// TwinCAT 3 PLC project utils
// Title: ESO ELT Utility Library
// Company: ESO
// Author: Mario Kiekebusch
// ProjectVersion: 0.0.0.2
// Description: ELT - Library provide general purpose utilities.
// ProgramVersion: 3.1.4023.0
// libraries:
//   ESO LDC Common Library, * (ESO)
//   ESO LDC Timer Library, * (ESO)
//   ESO MUDPI Library, * (ESO)
//   Tc2_Standard, * (Beckhoff Automation GmbH)
//   Tc2_System, * (Beckhoff Automation GmbH)
//   Tc2_Utilities, * (Beckhoff Automation GmbH)
//   Tc3_EventLogger, * (Beckhoff Automation GmbH)
//   Tc3_Module, * (Beckhoff Automation GmbH)
//   VisuDialogs, * (System)
// project tree:
//   DUTs/Structures/ T_EVENTLOG_PAYLOAD.TcDUT, T_EVENT_PUB_ELEM.TcDUT, T_IP_ADDRESS.TcDUT, T_PACKET_INFO.TcDUT, T_UDP_INFO.TcDUT
//   / GlobalTextList.TcGTLO, PlcTask.TcTTO, Visualization Manager.TcVMO (not stored)
//   GVLs/ GVL.TcGVL
//   POUs/ FB_DataSetFifo.TcPOU, FB_EVENT_LISTENER.TcPOU, FB_MUDPI_RECEIVER.TcPOU, FB_MUDPI_SENDER.TcPOU, FB_SAMPLE_LISTENER.TcPOU, MAIN.TcPOU
//   Version/ Global_Version.TcGVL
//   VISUs/Templates/ GUI_TEMPLATE_MUDPI_RECEIVER.TcVIS, GUI_TEMPLATE_MUDPI_SENDER.TcVIS
// real-time tasks:
//   TASK PlcTask: cycle T#10ms, priority 20, ADS port 350

CONFIGURATION utils
    RESOURCE PLC ON TwinCAT3
        TASK PlcTask(INTERVAL := T#10ms, PRIORITY := 20);
        PROGRAM MAIN WITH PlcTask : MAIN;
    END_RESOURCE
END_CONFIGURATION

// ---- DUTs/Structures/T_EVENTLOG_PAYLOAD.TcDUT
TYPE T_EVENTLOG_PAYLOAD :
STRUCT
	{attribute 'TcEncoding':='UTF-8'}
	source : STRING(80) := ''; 
	severity : INT := 0; 
	{attribute 'TcEncoding':='UTF-8'}
	text: STRING(255) := '';
	timestamp: ULINT;
END_STRUCT
END_TYPE

// ---- DUTs/Structures/T_EVENT_PUB_ELEM.TcDUT
TYPE T_EVENT_PUB_ELEM :
STRUCT
	fbEventText: FB_RequestEventText;
	bTextRequest: BOOL := FALSE;
	payload: T_EVENTLOG_PAYLOAD;
END_STRUCT
END_TYPE

// ---- DUTs/Structures/T_IP_ADDRESS.TcDUT
TYPE T_IP_ADDRESS :
UNION
	ipAdrInternal : UDINT;
	ipAdr : ARRAY[0..3] OF BYTE;
END_UNION
END_TYPE

// ---- DUTs/Structures/T_PACKET_INFO.TcDUT
TYPE T_PACKET_INFO :
STRUCT
	topicId: UDINT; 
	componentId: UINT; // counter the number of times the diagnostic data was sent.
	sampleId: UDINT; 
	frameId: UINT;
	numFrames: UINT;
	version: UINT;
	appTag: UINT;
	timestamp: LREAL;
	payloadSize: UINT;	
	size: UINT;
	valid: BOOL;
END_STRUCT
END_TYPE

// ---- DUTs/Structures/T_UDP_INFO.TcDUT
TYPE T_UDP_INFO :
STRUCT
	bDriverInitialization: BOOL; // Indication of whether the realtime driver is properly initialized.  
	nReceivedPackets: UDINT; // counter the number of times the diagnostic data was sent.
	uSenderAddress: T_IP_ADDRESS;
	ipv4Adr : T_IPv4Addr := '';
	lrNotification: LREAL; // timestamp of the last sent
	sNotification: STRING;
END_STRUCT
END_TYPE

// ---- GVLs/GVL.TcGVL
VAR_GLOBAL CONSTANT
	MAX_BUFFER_SIZE : UDINT := 35000;
	MAX_EVENTS_SIZE : INT := 100;
END_VAR

// ---- Version/Global_Version.TcGVL
{attribute 'TcGenerated'}
{attribute 'no-analysis'}
{attribute 'linkalways'}
// This function has been automatically generated from the project information.
VAR_GLOBAL CONSTANT
	{attribute 'const_non_replaced'}
	stLibVersion_ESO_ELT_Utility_Library : ST_LibVersion := (iMajor := 0, iMinor := 0, iBuild := 0, iRevision := 2, nFlags := 0, sVersion := '0.0.0.2');
END_VAR

// ---- POUs/MAIN.TcPOU
PROGRAM MAIN
VAR
END_VAR

END_PROGRAM

// ---- POUs/FB_DataSetFifo.TcPOU
FUNCTION_BLOCK FB_DataSetFifo
VAR_INPUT
	bOverwrite	: BOOL;
	in 			: T_EVENTLOG_PAYLOAD;
END_VAR
VAR_OUTPUT
	bOk			: BOOL;
	nCount		: UDINT;
	nLoad		: UDINT;
	out			: T_EVENTLOG_PAYLOAD;
END_VAR
VAR
	arrBuffer 	: ARRAY[0..MAX_BUFFER_SIZE] OF BYTE; (* Buffer memory used by FB_MemRingBuffer function block *)
	fbBuffer	: FB_MemRingBuffer;
	dataset_size: UDINT;
END_VAR

;

ACTION A_Add:
fbBuffer.A_AddTail( pWrite:= ADR( in ),
					cbWrite:= SIZEOF( in ),
					pBuffer:= ADR( arrBuffer ),
					cbBuffer:= SIZEOF( arrBuffer ),
					bOk=> bOk,
					nCount => nCount );


IF NOT bOk THEN (* overflow ? *)
	IF bOverwrite THEN
		fbBuffer.A_RemoveHead(); (* remove one oldest entry *)

		fbBuffer.A_AddTail( bOk => bOk, nCount => nCount );
	END_IF
END_IF


dataset_size := SIZEOF(in);
nLoad := (fbBuffer.cbSize * 100) / MAX_BUFFER_SIZE;
END_ACTION

ACTION A_Get:
fbBuffer.A_GetHead( pRead:= ADR( out ),
					cbRead:= SIZEOF( out ),
					pBuffer:= ADR( arrBuffer ),
					cbBuffer:= SIZEOF( arrBuffer ),
					bOk=> bOk,
					nCount => nCount );

nLoad := (fbBuffer.cbSize * 100) / MAX_BUFFER_SIZE;
END_ACTION

ACTION A_Remove:
fbBuffer.A_RemoveHead( 	pRead:= ADR( out ),
						cbRead:= SIZEOF( out ),
						pBuffer:= ADR( arrBuffer ),
						cbBuffer:= SIZEOF( arrBuffer ),
						bOk=> bOk,
						nCount => nCount );

nLoad := (fbBuffer.cbSize * 100) / MAX_BUFFER_SIZE;
END_ACTION

ACTION A_Reset:
MEMSET( ADR( arrBuffer ), 0, SIZEOF( arrBuffer ) ); (* reset (optional) internal buffer *)

fbBuffer.A_Reset( 	bOk=> bOk,
					nCount => nCount );

nLoad := (fbBuffer.cbSize * 100) / MAX_BUFFER_SIZE;
END_ACTION

METHOD IsEmpty : BOOL
VAR_INPUT
END_VAR
IF nCount > 0 THEN
	IsEmpty := FALSE;
	RETURN;
END_IF

IsEmpty := TRUE;
return;
END_METHOD

METHOD Size : UDINT
VAR_INPUT
END_VAR
Size := nCount;
END_METHOD

END_FUNCTION_BLOCK

// ---- POUs/FB_EVENT_LISTENER.TcPOU
FUNCTION_BLOCK FB_EVENT_LISTENER
VAR_INPUT
	refFbEventFilter  : REFERENCE TO FB_TcEventFilter; 
	refFbTime:  REFERENCE TO FB_TIME;
END_VAR
VAR_OUTPUT
END_VAR
VAR
	hr : HRESULT;
	
	bSubscribe : BOOL := TRUE;
	bSubscribed : BOOL;
	bUnSubscribe : BOOL;
	
	fbMessageListener : FB_SAMPLE_LISTENER;
	Message: INT;
	
END_VAR

fbMessageListener.CustomExecute(refFbTime); // retrieve messages and its texts


IF bSubscribe THEN 
	bSubscribe := FALSE;
	hr := fbMessageListener.Subscribe2(refFbEventFilter); //subscribe to retrieve defined events
	IF SUCCEEDED(hr) THEN	
		bSubscribed := TRUE;
	END_IF
END_IF 

IF bUnSubscribe THEN 
	bUnSubscribe := FALSE;
	hr := fbMessageListener.Unsubscribe();
	IF SUCCEEDED(hr) THEN	
		bSubscribed := FALSE;
	END_IF
END_IF

END_FUNCTION_BLOCK

// ---- POUs/FB_SAMPLE_LISTENER.TcPOU
FUNCTION_BLOCK FB_SAMPLE_LISTENER EXTENDS FB_ListenerBase2
VAR_INPUT
END_VAR
VAR_OUTPUT
END_VAR
VAR
	sJsonAttribute : STRING (10000);	
	hr : HRESULT;
	
	nCntMessagesSent : INT;
	nCntAlarmsRaised : INT;
	nCntAlarmsConfirmed : INT;
	nCntAlarmsCleared : INT;
	
	fbSender: FB_MUDPI_SENDER;
	arrEvents : ARRAY[0..MAX_EVENTS_SIZE] OF T_EVENT_PUB_ELEM;
	nCntEventReceived : INT := 0;
	fbFifo 		: FB_DataSetFifo := ( bOverwrite := TRUE );
	newEntry	: T_EVENTLOG_PAYLOAD;
	oldEntry	: T_EVENTLOG_PAYLOAD;
	bSuccess	: BOOL;
	nCount		: UDINT;
	nLoad		: UDINT;
	nWaitCounter : UDINT := 0;
END_VAR

METHOD CustomExecute : HRESULT
VAR_INPUT
	refFbTime:  REFERENCE TO FB_TIME;
END_VAR

VAR
	hr : HRESULT;
	counter: INT := 0;
END_VAR
hr := SUPER^.Execute(); //retrieve events
fbSender();
(* Go through the list of buffers to check if there new events *)
FOR counter := 0 TO MAX_EVENTS_SIZE BY 1 DO
	IF arrEvents[counter].bTextRequest THEN
		IF arrEvents[counter].fbEventText.bError THEN
			arrEvents[counter].payload.text := 'Error';
			arrEvents[counter].bTextRequest := FALSE;
			fbFifo.A_Add(	in := arrEvents[counter].payload, bOk=>bSuccess, nCount=> nCount, nLoad => nLoad );
		ELSIF NOT arrEvents[counter].fbEventText.bBusy THEN
			arrEvents[counter].fbEventText.GetString(arrEvents[counter].payload.text, SIZEOF(arrEvents[counter].payload.text));
			arrEvents[counter].bTextRequest := FALSE;
			(* add new entry to the fifo *)
			fbFifo.A_Add(	in := arrEvents[counter].payload, bOk=>bSuccess, nCount=> nCount, nLoad => nLoad );
		END_IF
	END_IF
END_FOR

// Forces to send one log per every ten cycles.
// Due to the asynchronous nature of the TC Event Logging, sending the logs faster has 
// shown some problems. 
IF NOT fbFifo.IsEmpty() THEN
	nWaitCounter := nWaitCounter + 1;
	IF nWaitCounter > 10 THEN
		(* remove oldest entry from them ring buffer*)
		fbFifo.A_Remove( out => oldEntry, bOk => bSuccess, nCount => nCount, nLoad => nLoad );
		IF bSuccess THEN
			(* Send log info *)
			fbSender.SetTimestamp(refFbTime.GetMudpiTime());
			fbSender.SetMudpiPayload(ADR(oldEntry), SIZEOF(oldEntry));
			fbSender.SendData();
			(* Reset counter *)
			nWaitCounter := 0;
		END_IF
	END_IF
END_IF 



CustomExecute:= hr;
END_METHOD

METHOD OnAlarmCleared : HRESULT
VAR_INPUT
	fbEvent : REFERENCE TO FB_TcEvent;
END_VAR
nCntAlarmsCleared := nCntAlarmsCleared + 1;

OnAlarmCleared := S_OK; // in order to receive more callbacks (Set <> S_OK in order to cancel the callbacks for this program cycle.)
END_METHOD

METHOD OnAlarmConfirmed : HRESULT
VAR_INPUT
	fbEvent : REFERENCE TO FB_TcEvent;
END_VAR
nCntAlarmsConfirmed := nCntAlarmsConfirmed + 1;

OnAlarmConfirmed := S_OK; // in order to receive more callbacks (Set <> S_OK in order to cancel the callbacks for this program cycle.)
END_METHOD

METHOD OnAlarmRaised : HRESULT
VAR_INPUT
	fbEvent : REFERENCE TO FB_TcEvent;
END_VAR
hr := fbEvent.GetJsonAttribute(sJsonAttribute, SIZEOF(sJsonAttribute));
nCntAlarmsRaised := nCntAlarmsRaised + 1;

OnAlarmRaised := S_OK; // in order to receive more callbacks (Set <> S_OK in order to cancel the callbacks for this program cycle.)
END_METHOD

METHOD OnMessageSent : HRESULT
VAR_INPUT
	fbEvent : REFERENCE TO FB_TcEvent;
END_VAR

VAR
	payload: T_EVENTLOG_PAYLOAD;
	fbRequestEventText : FB_RequestEventText;
END_VAR
hr := fbEvent.GetJsonAttribute(sJsonAttribute, SIZEOF(sJsonAttribute));

(* Store events in an array since they could arrive in bursts *)
arrEvents[nCntEventReceived].bTextRequest :=  TRUE;
arrEvents[nCntEventReceived].payload.source := fbEvent.ipSourceInfo.sName;
arrEvents[nCntEventReceived].payload.severity := fbEvent.eSeverity;
arrEvents[nCntEventReceived].payload.timestamp := fbEvent.nTimestamp;
arrEvents[nCntEventReceived].fbEventText.Request(eventClass:=fbEvent.EventClass, nEventId:=fbEvent.nEventId, nLangId:=1033, ipArgs:=fbEvent.ipArguments );
arrEvents[nCntEventReceived].bTextRequest :=  TRUE;
nCntMessagesSent := nCntMessagesSent + 1;
nCntEventReceived := nCntEventReceived + 1;
(*
If number of events are bigger than the buffer size, start overiding 
The risk of loosing events is low since we have a ring buffer storing 
the events to be sent outside. 
*)
IF nCntEventReceived >= MAX_EVENTS_SIZE THEN
	nCntEventReceived := 0;
END_IF



OnMessageSent := S_OK; // in order to receive more callbacks (Set <> S_OK in order to cancel the callbacks for this program cycle.)
END_METHOD

END_FUNCTION_BLOCK

// ---- POUs/FB_MUDPI_SENDER.TcPOU
(*
    This function blocks aims to pack the EL6688 diagnostic data in MUDPI frames
    and transmit them to Time System using Beckhoffs realtime UDP driver (TF6311). 
    The user of this function blocks needs to do the following in order for the library to work correctly:
    - Initialize the library with configuration parameters
        - Destination IP-address (a multicast address)
        - Destination port
        - Source port
*)

{attribute 'c++_compatible'}
FUNCTION_BLOCK FB_MUDPI_SENDER IMPLEMENTS ITcIoUdpProtocolRecv
VAR_INPUT
		ipAddress : Tc2_System.T_IPv4Addr := '0.0.0.0';
		dest_port : UINT := 10000;
		local_port : UINT := 20000;
		instance_name: STRING := 'undefined';
END_VAR
VAR_OUTPUT
END_VAR
VAR
	(* TF6311 realtime driver parameters *)
    {attribute 'TcInitSymbol'}
    oid : OTCID;
    ipUdp : ITcIoUdpProtocol;
    nReceivedPackets : UINT;
    uLastReceivedIP : T_IP_ADDRESS;
    hrInit : HRESULT;
    hrSend : HRESULT; 
    bSuccessfulInitializationOfRealtimeDriver : BOOL := FALSE; // Indication of whether the realtime driver is properly initialized.
	bEnableSending : BOOL := FALSE; // Indication of whether the sender is active or not.
	
	mudpiPacket : ESO_MUDPI.FB_MudpiPacket(topicId := 300, componentId := 5);
	packet_info : T_PACKET_INFO;
	
	  (* Transmission/communication parameters *)
	_destinationIpAddressString : Tc2_System.T_IPv4Addr;
    _destinationIpAddress : UDINT; // Destination address for the data
    _destinationPort : UINT; // Destination port for the data
    _sourcePort : UINT; // Source port of the data
	
	sLibVersion:	   STRING	:= 'UNKNOWN'; // Library version
	
END_VAR

(*
_destinationIpAddressString := ipAddress;
_destinationPort := dest_port;
_sourcePort := local_port;
*)

IF ipUdp <> 0 THEN
	ipUdp.CheckReceived();
END_IF

UpdateMudpiPacket();

METHOD FB_exit : BOOL
VAR_INPUT
    bInCopyCode : BOOL; // if TRUE, the exit method is called for exiting an instance that is copied afterwards (online change).
END_VAR
IF NOT bInCopyCode THEN // no online change
    IF ipUdp <> 0 THEN
        //ipUdp.UnregisterReceiver(nUdpPort); // Shutdown
        //ipUdp.UnregisterReceiver(nUdpPort); // Shutdown
        FW_SafeRelease(ADR(ipUdp));
        FB_exit := TRUE;
    END_IF
END_IF
END_METHOD

METHOD FB_init : BOOL
VAR_INPUT
    bInitRetains : BOOL; // if TRUE, the retain variables are initialized (warm start / cold start)
    bInCopyCode : BOOL;  // if TRUE, the instance afterwards gets moved into the copy code (online change)
END_VAR

sLibVersion := stLibVersion_ESO_ELT_Utility_Library.sVersion;
_destinationIpAddressString := ipAddress;
_destinationPort := dest_port;
_sourcePort := local_port;

IF NOT bInCopyCode THEN // no online change
	IF ipUdp = 0 AND oid <> 0 THEN
	    hrInit := FW_ObjMgr_GetObjectInstance(	oid:=oid, 
											iid:=TC_GLOBAL_IID_LIST.IID_ITcIoUdpProtocol, 
											pipUnk:=ADR(ipUdp) );
		
		IF SUCCEEDED(hrInit) THEN 
			bSuccessfulInitializationOfRealtimeDriver := TRUE;
		(*
			IF  SUCCEEDED(ipUdp.RegisterReceiver(nUdpPort, THIS^)) THEN //open port
				FB_init := TRUE;
			ELSE 
				FB_init := FALSE; 
				FW_SafeRelease(ADR(ipUdp));
			END_IF
			*)
		END_IF
		
	ELSIF oid = 0 THEN 
		FB_init := FALSE; 
		hrInit := ERR_INVALID_PARAM; 				
	END_IF
END_IF
END_METHOD

METHOD FB_reinit : BOOL
IF (ipUdp <> 0) THEN
    //ipUdp.RegisterReceiver(nUdpPort, THIS^);
    //ipUdp.RegisterReceiver(nUdpPort, THIS^);
    FB_reinit := TRUE;
END_IF
END_METHOD

{attribute 'c++_compatible'}
{attribute 'minimal_input_size' := '4'}
{attribute 'pack_mode' := '4'}
METHOD ReceiveData : HRESULT
VAR_INPUT
	ipAddr	: UDINT;
	udpDestPort	: UINT;
	udpSrcPort	: UINT;
	nData	: UDINT;
	pData	: PVOID;
	pVlan	: POINTER TO ETYPE_VLAN_HEADER := 0;
END_VAR
nReceivedPackets := nReceivedPackets + 1;
uLastReceivedIP.ipAdrInternal := ipAddr;
END_METHOD

(*
    This method carry out the sending of the diagnostic data using the Ethernet network driver.
    The parameters are the array of data to be sent and the timestamp that is required by
	the MUDPI protocol.
*)

METHOD SendData : HRESULT
VAR_INPUT
END_VAR
	 
VAR
	
END_VAR

_DestinationIpAddress := F_IpAddress2Integer(_destinationIpAddressString);
IF ipUdp <> 0 AND bSuccessfulInitializationOfRealtimeDriver = TRUE AND bEnableSending THEN
						   
		// Send Data via UDP
    hrSend := ipUdp.SendData(ipDestAddr := _DestinationIpAddress,
                             udpDestPort := _DestinationPort,
                             udpSrcPort := _SourcePort,
                             nData := mudpiPacket.Size(),
                             pData := mudpiPacket.Data(),
                             bCalcUdpCheckSum := FALSE,
                             pVlan := 0);
    IF SUCCEEDED(hrSend) THEN
        mudpiPacket.IncreaseSampleId();
	END_IF
END_IF


SendData:= hrSend;
END_METHOD

METHOD PUBLIC SetMudpiPayload : BOOL
VAR_INPUT
    payload : POINTER TO BYTE;
    payloadSize : UINT;
END_VAR
SetMudpiPayload := mudpiPacket.SetPayload(payload, payloadSize);
END_METHOD

METHOD PUBLIC SetPacketInfo
VAR_INPUT
    TopicId : UDINT; // MUDPI Topic identity
    ComponentId : UINT; // MUDPI component identity
	Timestamp: LREAL := 0;
END_VAR
packet_info.topicId := TopicId;
packet_info.componentId := ComponentId;
packet_info.timestamp := Timestamp;
UpdateMudpiPacket();
END_METHOD

METHOD PUBLIC SetTimestamp
VAR_INPUT
	Timestamp: LREAL;
END_VAR
packet_info.timestamp := Timestamp;
mudpiPacket.SetTimestamp(packet_info.timestamp);
END_METHOD

{attribute 'c++_compatible'}
{attribute 'minimal_input_size' := '4'}
{attribute 'pack_mode' := '4'}
METHOD TcAddRef : UDINT
END_METHOD

{attribute 'object_name' := 'TcQueryInterface'}
{attribute 'c++_compatible'}
{attribute 'signature_flag' := '33554688'}
{attribute 'pack_mode' := '4'}
{attribute 'show'}
{attribute 'minimal_input_size' := '4'}
METHOD TcQueryInterface : HRESULT
VAR_INPUT
	iid	: REFERENCE TO IID;
	pipItf	: POINTER TO PVOID;
END_VAR
VAR
	ipUdpRecv : ITcIoUdpProtocolRecv;
	ipUnknown : ITcUnknown;	
END_VAR
IF GuidsEqual(ADR(iid), ADR(TC_GLOBAL_IID_LIST.IID_ITcIoUdpProtocolRecv)) THEN
	ipUdpRecv := THIS^; // cast to interface pointer
	pipItf^ := ITCUNKNOWN_TO_PVOID(ipUdpRecv);
	TcAddRef();
	TcQueryInterface := S_OK;
ELSIF GuidsEqual(ADR(iid), ADR(TC_GLOBAL_IID_LIST.IID_ITcUnknown)) THEN
	ipUnknown := THIS^; // cast to interface pointer
	pipItf^ := ITCUNKNOWN_TO_PVOID(ipUnknown);
	TcAddRef();
	TcQueryInterface := S_OK;
ELSE
	TcQueryInterface := E_HRESULTAdsErr.NOINTERFACE ; //Call super if this fb extends some other
END_IF
END_METHOD

{attribute 'c++_compatible'}
{attribute 'minimal_input_size' := '4'}
{attribute 'pack_mode' := '4'}
METHOD TcRelease : UDINT
END_METHOD

METHOD PUBLIC UpdateMudpiPacket
VAR_INPUT
END_VAR

mudpiPacket.SetTopicId(packet_info.topicId);
mudpiPacket.SetComponentId(packet_info.componentId);
mudpiPacket.SetTimestamp(packet_info.timestamp);
END_METHOD

END_FUNCTION_BLOCK

// ---- POUs/FB_MUDPI_RECEIVER.TcPOU
(*
    This function blocks aims to CCS data coming in MUDPI frames.
    It uses the Beckhoff realtime UDP driver (TF6311). 
    The user of this function blocks needs to do the following in order for the library to work correctly:
    - Initialize the library with configuration parameters
        - Source port
*)

{attribute 'c++_compatible'}
FUNCTION_BLOCK FB_MUDPI_RECEIVER IMPLEMENTS ITcIoUdpProtocolRecv
VAR_INPUT
	port : UINT := 10000;
	instance_name: STRING := 'undefined';
END_VAR
VAR_OUTPUT
END_VAR
VAR
	(* TF6311 realtime driver parameters *)
    {attribute 'TcInitSymbol'}
    oid : OTCID;
    ipUdp : ITcIoUdpProtocol;
	nUdpPort : UINT := port;
    nReceivedPackets : UINT;
    uLastReceivedIP : T_IP_ADDRESS;
    hrInit : HRESULT;
    bSuccessfulInitializationOfRealtimeDriver : BOOL := FALSE; 
	(* Data/contents parameters *)
    mudpiPacket : ESO_MUDPI.FB_MudpiPacket(topicId := 300, componentId := 5);
	packet_info : T_PACKET_INFO;
	udp_info: T_UDP_INFO;
	sLibVersion:	   STRING	:= 'UNKNOWN'; // Library version
   

	
END_VAR

IF ipUdp <> 0 THEN
	ipUdp.CheckReceived();
END_IF

METHOD FB_exit : BOOL
VAR_INPUT
    bInCopyCode : BOOL; // if TRUE, the exit method is called for exiting an instance that is copied afterwards (online change).
END_VAR
IF NOT bInCopyCode THEN // no online change
    IF ipUdp <> 0 THEN
        //ipUdp.UnregisterReceiver(nUdpPort); // Shutdown
        ipUdp.UnregisterReceiver(nUdpPort); // Shutdown
        FW_SafeRelease(ADR(ipUdp));
        FB_exit := TRUE;
    END_IF
END_IF
END_METHOD

METHOD FB_init : BOOL
VAR_INPUT
    bInitRetains : BOOL; // if TRUE, the retain variables are initialized (warm start / cold start)
    bInCopyCode : BOOL;  // if TRUE, the instance afterwards gets moved into the copy code (online change)
END_VAR

sLibVersion := stLibVersion_ESO_ELT_Utility_Library.sVersion;

IF NOT bInCopyCode THEN // no online change
	IF ipUdp = 0 AND oid <> 0 THEN
	    hrInit := FW_ObjMgr_GetObjectInstance(	oid:=oid, 
											iid:=TC_GLOBAL_IID_LIST.IID_ITcIoUdpProtocol, 
											pipUnk:=ADR(ipUdp) );
		IF SUCCEEDED(hrInit) THEN 
			IF  SUCCEEDED(ipUdp.RegisterReceiver(nUdpPort, THIS^)) THEN //open port
				FB_init := TRUE;
				udp_info.bDriverInitialization := TRUE;
				(*bSuccessfulInitializationOfRealtimeDriver := TRUE;*)
			ELSE 
				FB_init := FALSE; 
				FW_SafeRelease(ADR(ipUdp));
			END_IF
		END_IF
	ELSIF oid = 0 THEN 
		FB_init := FALSE; 
		hrInit := ERR_INVALID_PARAM; 				
	END_IF
END_IF
END_METHOD

METHOD FB_reinit : BOOL
IF (ipUdp <> 0) THEN
    //ipUdp.RegisterReceiver(nUdpPort, THIS^);
    ipUdp.RegisterReceiver(nUdpPort, THIS^);
    FB_reinit := TRUE;
END_IF
END_METHOD

METHOD PUBLIC GetMudpiPayload : POINTER TO BYTE
GetMudpiPayload := mudpiPacket.GetPayload();
END_METHOD

METHOD PUBLIC GetMudpiPayloadSize : UINT
GetMudpiPayloadSize := mudpiPacket.GetPayloadSize();
END_METHOD

METHOD PUBLIC GetTimestamp : LREAL
VAR_INPUT	
END_VAR

GetTimestamp := packet_info.timestamp;
END_METHOD

METHOD PRIVATE IpAddressStringToInteger : UDINT
VAR_INPUT
    IpAddress : Tc2_System.T_IPv4Addr;
END_VAR
VAR
    IpAddressArray : Tc2_System.T_IPv4AddrArr;
    IpAddressInteger : UDINT;
END_VAR
IpAddressArray := Tc2_System.F_ScanIPv4AddrIds(sIPv4 := IpAddress);
IpAddressInteger := LREAL_TO_UDINT(IpAddressArray[0] * EXPT(256, 3) +
                                   IpAddressArray[1] * EXPT(256, 2) +
                                   IpAddressArray[2] * EXPT(256, 1) +
                                   IpAddressArray[3]);

IpAddressStringToInteger := IpAddressInteger;
END_METHOD

METHOD PRIVATE IpIntegerToAddressString : Tc2_System.T_IPv4Addr
VAR_INPUT
    IpAddress : T_IP_ADDRESS;
END_VAR
VAR
    IpAddressArray : Tc2_System.T_IPv4AddrArr;
	
END_VAR



IpAddressArray[3] := IpAddress.ipAdr[0];
IpAddressArray[2] := IpAddress.ipAdr[1];
IpAddressArray[1] := IpAddress.ipAdr[2];
IpAddressArray[0] := IpAddress.ipAdr[3];

IpIntegerToAddressString := F_CreateIPv4Addr( IpAddressArray );
END_METHOD

{attribute 'c++_compatible'}
{attribute 'minimal_input_size' := '4'}
{attribute 'pack_mode' := '4'}
METHOD ReceiveData : HRESULT
VAR_INPUT
	ipAddr	: UDINT;
	udpDestPort	: UINT;
	udpSrcPort	: UINT;
	nData	: UDINT;
	pData	: PVOID;
	pVlan	: POINTER TO ETYPE_VLAN_HEADER := 0;
END_VAR
VAR
	tmp: LREAL;
END_VAR

VAR CONSTANT
	UNIX_OFFSET_MICROSEC: ULINT := DATE_TO_ULINT(DATE#2000-01-01) * 10#1000_000;
END_VAR
(*
nReceivedPackets := nReceivedPackets + 1;
uLastReceivedIP.ipAdrInternal := ipAddr;
memset(ADR(buffer), 0, SIZEOF(buffer));
memcpy(ADR(buffer), pData, nData);
*)
udp_info.nReceivedPackets := udp_info.nReceivedPackets + 1;
udp_info.uSenderAddress.ipAdrInternal := ipAddr;
udp_info.ipv4Adr := IpIntegerToAddressString(udp_info.uSenderAddress);

mudpiPacket.Initialize(inputData := pData,
                  size := UDINT_TO_UINT(nData));
packet_info.topicId := mudpiPacket.GetTopicId();
packet_info.componentId := mudpiPacket.GetComponentId();
packet_info.appTag := mudpiPacket.GetApplicationTag();
packet_info.version := mudpiPacket.GetVersion();
packet_info.frameId := mudpiPacket.GetFrameId();
packet_info.sampleId := mudpiPacket.GetSampleId();
packet_info.size := UDINT_TO_UINT(nData);
packet_info.payloadSize := mudpiPacket.GetPayloadSize();
packet_info.timestamp := mudpiPacket.GetTimestamp();
packet_info.valid := ValidatePacket();
END_METHOD

{attribute 'c++_compatible'}
{attribute 'minimal_input_size' := '4'}
{attribute 'pack_mode' := '4'}
{warning 'add method implementation'}
METHOD TcAddRef : UDINT
END_METHOD

{attribute 'object_name' := 'TcQueryInterface'}
{attribute 'c++_compatible'}
{attribute 'signature_flag' := '33554688'}
{attribute 'pack_mode' := '4'}
{attribute 'show'}
{attribute 'minimal_input_size' := '4'}
METHOD TcQueryInterface : HRESULT
VAR_INPUT
	iid	: REFERENCE TO IID;
	pipItf	: POINTER TO PVOID;
END_VAR
VAR
	ipUdpRecv : ITcIoUdpProtocolRecv;
	ipUnknown : ITcUnknown;	
END_VAR
IF GuidsEqual(ADR(iid), ADR(TC_GLOBAL_IID_LIST.IID_ITcIoUdpProtocolRecv)) THEN
	ipUdpRecv := THIS^; // cast to interface pointer
	pipItf^ := ITCUNKNOWN_TO_PVOID(ipUdpRecv);
	TcAddRef();
	TcQueryInterface := S_OK;
ELSIF GuidsEqual(ADR(iid), ADR(TC_GLOBAL_IID_LIST.IID_ITcUnknown)) THEN
	ipUnknown := THIS^; // cast to interface pointer
	pipItf^ := ITCUNKNOWN_TO_PVOID(ipUnknown);
	TcAddRef();
	TcQueryInterface := S_OK;
ELSE
	TcQueryInterface := E_HRESULTAdsErr.NOINTERFACE ; //Call super if this fb extends some other
END_IF
END_METHOD

{attribute 'c++_compatible'}
{attribute 'minimal_input_size' := '4'}
{attribute 'pack_mode' := '4'}
{warning 'add method implementation'}
METHOD TcRelease : UDINT
END_METHOD

(*
    This method verifies, if the checksum of a MUDPI packet is correct.
    TRUE = Checksum does match the content of the packet, FALSE = checksum does not match.
*)
METHOD PUBLIC ValidatePacket : BOOL
VAR
    checksum1 : UINT;
    checksum2 : UINT;
END_VAR

ValidatePacket := mudpiPacket.VerifyPacket();
END_METHOD

END_FUNCTION_BLOCK

// ---- GlobalTextList.TcGTLO
TEXTLIST GlobalTextList
  577 = '%s'
  1009 = 'App Tag'
  337 = 'CCS library ver. %s'
  746 = 'Component ID'
  1119 = 'Dest Port'
  743 = 'Disable'
  1047 = 'Disable Diagnostics'
  536 = 'Enable'
  742 = 'Enable Diagnostics'
  537 = 'Enabled'
  568 = 'Ethernet driver initialization'
  963 = 'Frame ID '
  787 = 'Instance: %s'
  505 = 'IP address'
  43 = 'Packet Counter'
  703 = 'Packet Info'
  1057 = 'Payload size'
  115 = 'RED - False\nGREEN - True'
  1156 = 'Sample ID'
  263 = 'Size'
  749 = 'Time used for Simulation. \nPress "Copy UTC" or "Copy Local" button to get the time in correct format and then modify it for your needs.'
  184 = 'Timestamp'
  671 = 'Topic ID'
  322 = 'UDP Receiver'
  1124 = 'UDP Sender'
  907 = 'Version'
  356 = 'WHITE - Disabled\nGREEN - Enabled'
END_TEXTLIST

// ---- VISUs/Templates/GUI_TEMPLATE_MUDPI_RECEIVER.TcVIS
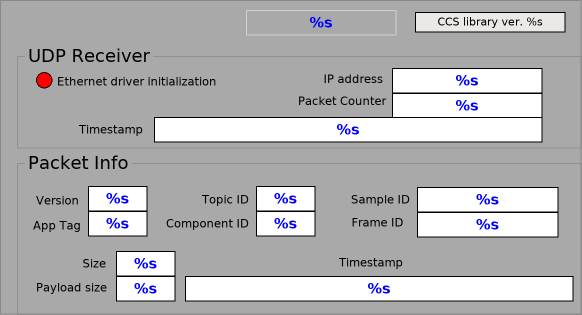
VISUALIZATION GUI_TEMPLATE_MUDPI_RECEIVER  // 582x315
VAR_INPUT
	m_DeviceName : STRING;
END_VAR
VAR_IN_OUT
	m_Instance : FB_MUDPI_RECEIVER;
END_VAR
    GroupBox (17,48 565x100), "UDP Receiver"
        Rectangle (375,20 150x25), "%s", text variable: m_Instance.udp_info.ipv4Adr
            OnMouseDown: write the text variable via Edit
        Label (285,18 84x26), "IP address"
        Label (37,19 240x29), "Ethernet driver initialization"
        Ellipse (19,24 16x16), tooltip "RED - False GREEN - True", colour toggle: m_Instance.udp_info.bDriverInitialization
        Label (265,40 107x26), "Packet Counter"
        Rectangle (375,45 150x25), "%s", text variable: m_Instance.udp_info.nReceivedPackets
            OnMouseDown: write the text variable via Edit
        Rectangle (137,69 388x25), "%s", tooltip "Time used for Simulation. Press "Copy UTC" or "Copy Local" button to get the time in correct format and then modify it for your needs.", text variable: m_Instance.udp_info.sNotification
            OnMouseDown: write the text variable via Default
        Label (56,70 76x23), "Timestamp"
    Rectangle (246,10 150x25), "%s", text variable: m_Instance.instance_name
    Rectangle (415,12 150x20), "CCS library ver. %s", text variable: m_Instance.sLibVersion
    GroupBox (17,155 565x160), "Packet Info"
        Rectangle (71,31 59x25), "%s", text variable: m_Instance.packet_info.version
            OnMouseDown: write the text variable via Edit
        Rectangle (71,56 59x25), "%s", text variable: m_Instance.packet_info.appTag
            OnMouseDown: write the text variable via Edit
        Label (6,31 59x29), "Version"
        Label (6,56 61x29), "App Tag"
        Label (329,30 67x29), "Sample ID"
        Rectangle (400,32 141x25), "%s", text variable: m_Instance.packet_info.sampleId
            OnMouseDown: write the text variable via Edit
        Rectangle (239,31 59x25), "%s", text variable: m_Instance.packet_info.topicId
            OnMouseDown: write the text variable via Edit
        Label (176,30 59x29), "Topic ID"
        Label (148,54 87x29), "Component ID"
        Rectangle (239,56 59x25), "%s", text variable: m_Instance.packet_info.componentId
            OnMouseDown: write the text variable via Edit
        Rectangle (400,57 141x25), "%s", text variable: m_Instance.packet_info.frameId
            OnMouseDown: write the text variable via Edit
        Label (304,53 89x29), "Frame ID"
        Label (316,96 76x23), "Timestamp"
        Rectangle (168,121 388x25), "%s", tooltip "Time used for Simulation. Press "Copy UTC" or "Copy Local" button to get the time in correct format and then modify it for your needs.", text variable: m_Instance.packet_info.timestamp
            OnMouseDown: write the text variable via Default
        Label (25,94 67x29), "Size"
        Label (12,118 81x29), "Payload size"
        Rectangle (99,96 59x25), "%s", text variable: m_Instance.packet_info.size
            OnMouseDown: write the text variable via Edit
        Rectangle (99,121 59x25), "%s", text variable: m_Instance.packet_info.payloadSize
            OnMouseDown: write the text variable via Edit
END_VISUALIZATION

// ---- VISUs/Templates/GUI_TEMPLATE_MUDPI_SENDER.TcVIS
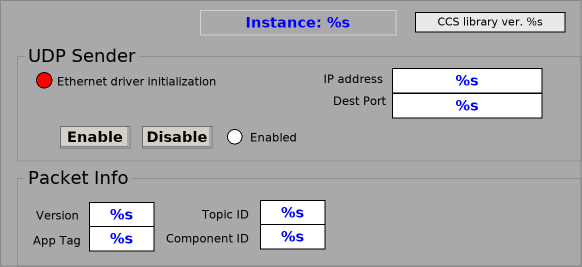
VISUALIZATION GUI_TEMPLATE_MUDPI_SENDER  // 582x267
VAR_INPUT
	m_DeviceName : STRING;
END_VAR
VAR_IN_OUT
	m_Instance : FB_MUDPI_SENDER;
END_VAR
    GroupBox (17,48 565x113), "UDP Sender"
        Rectangle (375,20 150x25), "%s", text variable: m_Instance._destinationIpAddressString
            OnMouseDown: write the text variable via Edit
        Label (285,18 84x26), "IP address"
        Label (37,19 240x29), "Ethernet driver initialization"
        Ellipse (19,24 16x16), tooltip "RED - False GREEN - True", colour toggle: m_Instance.bSuccessfulInitializationOfRealtimeDriver
        Label (265,40 107x26), "Dest Port"
        Rectangle (375,45 150x25), "%s", text variable: m_Instance._destinationPort
            OnMouseDown: write the text variable via Edit
        Button (43,78 70x22), "Enable", tooltip "Enable Diagnostics"
            OnMouseClick: execute { m_Instance.bEnableSending := TRUE; }
        Button (125,78 70x22), "Disable", tooltip "Disable Diagnostics"
            OnMouseClick: execute { m_Instance.bEnableSending := FALSE; }
        Label (230,75 61x29), "Enabled"
        Ellipse (210,81 15x15), tooltip "WHITE - Disabled GREEN - Enabled", colour toggle: m_Instance.bEnableSending
    Rectangle (200,10 196x25), "Instance: %s", text variable: m_Instance.instance_name
    Rectangle (415,12 150x20), "CCS library ver. %s", text variable: m_Instance.sLibVersion
    GroupBox (17,170 565x97), "Packet Info"
        Label (6,31 59x29), "Version"
        Label (6,56 61x29), "App Tag"
        Label (176,30 59x29), "Topic ID"
        Label (148,54 87x29), "Component ID"
        Rectangle (243,30 65x25), "%s", text variable: m_Instance.packet_info.topicId
            OnMouseDown: write the text variable via Edit
        Rectangle (243,54 65x25), "%s", text variable: m_Instance.packet_info.componentId
            OnMouseDown: write the text variable via Edit
        Rectangle (72,32 65x25), "%s", text variable: m_Instance.packet_info.version
            OnMouseDown: write the text variable via Edit
    Rectangle (89,226 65x25), "%s", text variable: m_Instance.packet_info.appTag
        OnMouseDown: write the text variable via Edit
END_VISUALIZATION
